FUNCTION_BLOCK Sensor_Notimplemented
VAR_INPUT
END_VAR
VAR_OUTPUT
END_VAR
VAR
END_VAR

END_FUNCTION_BLOCK

(* stored: Version 1.1.0.1, ProductVersion 3.1.4024.6
   POU Sensor_Notimplemented: Id {bf58be98-0551-4cb2-83fe-ff7fd445bd23}, SpecialFunc None *)
